Yaskawa INFORM job: ramp_standing_planes_program.JBI

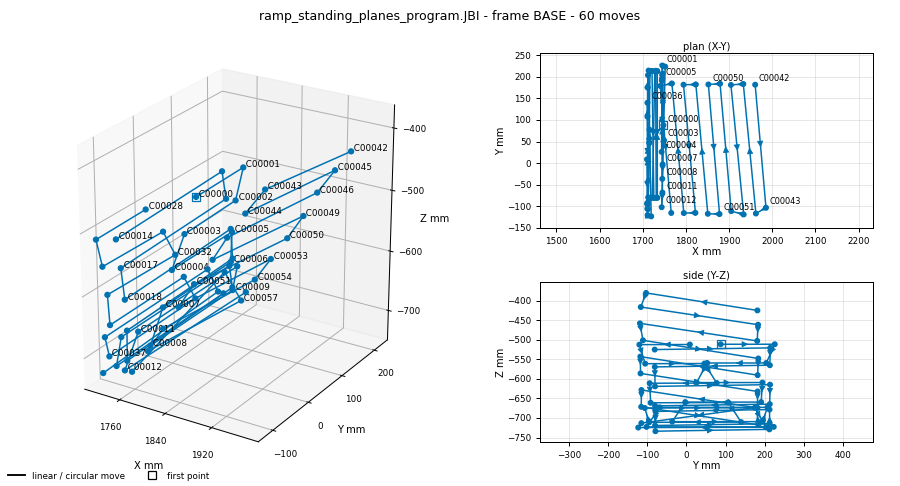
[picture p0: tool path of ramp_standing_planes_program.JBI in frame BASE, 60 of 65 moves have a stored position in this frame; points joined in program order, loops and branches not executed]
/JOB
//NAME ramp_standing_planes_program
//POS
///NPOS 60,0,60,0,0,0
///TOOL 0
///POSTYPE BASE
///RECTAN
///RCONF 0,0,0,0,0,0,0,0,0,0,0,0,0,0,0,0,0,0,0,0,0,0,0,0
C00000=1747.833676,87.707513,-511.371116,5.000000,-89.957822,175.000000
C00001=1745.440097,225.996535,-511.342791,5.000000,-89.957822,175.000000
C00002=1744.923440,204.207688,-559.299641,5.000000,-89.957822,175.000000
C00003=1749.154270,53.149469,-559.329393,5.000000,-89.957822,175.000000
C00004=1743.721814,26.039255,-609.339304,5.000000,-89.957822,175.000000
C00005=1744.348289,194.565765,-609.302177,5.000000,-89.957822,175.000000
C00006=1744.187925,191.095267,-659.303065,5.000000,-89.957822,175.000000
C00007=1746.082813,-2.901127,-659.343877,5.000000,-89.957822,175.000000
C00008=1745.263776,-36.374100,-709.351778,5.000000,-89.957822,175.000000
C00009=1745.079107,194.848338,-709.301607,5.000000,-89.957822,175.000000
C00010=1746.036638,207.361004,-672.695654,180.000000,-60.000000,0.000000
C00011=1745.574257,-68.103268,-672.755927,180.000000,-60.000000,0.000000
C00012=1743.877002,-102.062921,-722.764579,180.000000,-60.000000,0.000000
C00013=1752.018887,223.400139,-722.687777,180.000000,-60.000000,0.000000
C00014=1718.533268,-81.118931,-524.973339,5.000000,-87.037114,175.000000
C00015=1713.684878,214.380906,-520.671837,5.000000,-87.037114,175.000000
C00016=1721.540048,213.468866,-565.028354,5.000000,-87.037114,175.000000
C00017=1725.758225,-80.815821,-569.343755,5.000000,-87.037114,175.000000
C00018=1731.242809,-80.197878,-619.123216,5.000000,-87.037114,175.000000
C00019=1729.852338,213.811139,-614.665704,5.000000,-87.037114,175.000000
C00020=1733.681143,213.171353,-664.550241,5.000000,-87.037114,175.000000
C00021=1733.797506,-80.066986,-669.061826,5.000000,-87.037114,175.000000
C00022=1733.019581,-80.164547,-719.176447,5.000000,-87.037114,175.000000
C00023=1733.370862,212.848816,-714.644124,5.000000,-87.037114,175.000000
C00024=1727.945778,212.635262,-678.398521,180.000000,-60.000000,0.000000
C00025=1722.359725,-78.980421,-683.180255,180.000000,-60.000000,0.000000
C00026=1712.658875,-79.296819,-733.760083,180.000000,-60.000000,0.000000
C00027=1716.885173,212.264276,-729.049569,180.000000,-60.000000,0.000000
C00028=1709.955725,8.794869,-512.045023,5.000000,-89.491817,175.000000
C00029=1711.306908,-120.321693,-512.369923,5.000000,-89.491817,175.000000
C00030=1710.700045,-105.520124,-561.084797,5.000000,-89.491817,175.000000
C00031=1715.144631,46.230498,-560.649434,5.000000,-89.491817,175.000000
C00032=1715.725129,77.457805,-610.564946,5.000000,-89.491817,175.000000
C00033=1709.951896,-93.988220,-611.063481,5.000000,-89.491817,175.000000
C00034=1711.444659,-91.511088,-661.045915,5.000000,-89.491817,175.000000
C00035=1710.974292,107.455154,-660.530954,5.000000,-89.491817,175.000000
C00036=1710.807654,139.847878,-710.450052,5.000000,-89.491817,175.000000
C00037=1711.661647,-95.428769,-711.056349,5.000000,-89.491817,175.000000
C00038=1712.376345,-106.493392,-674.478476,180.000000,-60.000000,0.000000
C00039=1711.169902,174.896087,-673.754989,180.000000,-60.000000,0.000000
C00040=1712.211733,203.656058,-723.672846,180.000000,-60.000000,0.000000
C00041=1719.670531,-123.239544,-724.459608,180.000000,-60.000000,0.000000
C00042=1960.330006,181.614488,-424.835174,175.000000,-56.152488,-5.000000
C00043=1985.368889,-103.193855,-380.137392,175.000000,-56.152488,-5.000000
C00044=1962.016425,-116.674380,-416.148142,175.000000,-56.152488,-5.000000
C00045=1932.882821,183.234864,-461.360037,175.000000,-56.152488,-5.000000
C00046=1904.216477,181.050268,-502.826697,175.000000,-56.152488,-5.000000
C00047=1933.813388,-118.873277,-457.922429,175.000000,-56.152488,-5.000000
C00048=1904.866793,-111.166767,-501.336623,175.000000,-56.152488,-5.000000
C00049=1879.065944,183.890803,-547.736137,175.000000,-56.152488,-5.000000
C00050=1852.001340,182.186319,-590.380650,175.000000,-56.152488,-5.000000
C00051=1877.849575,-117.893555,-542.928603,175.000000,-56.152488,-5.000000
C00052=1850.711806,-117.345247,-586.010425,175.000000,-56.152488,-5.000000
C00053=1823.000964,182.124997,-632.081707,175.000000,-56.152488,-5.000000
C00054=1794.417051,181.587415,-673.959238,175.000000,-56.152488,-5.000000
C00055=1822.009926,-115.041980,-628.422180,175.000000,-56.152488,-5.000000
C00056=1795.135163,-115.591042,-671.443463,175.000000,-56.152488,-5.000000
C00057=1767.615554,184.356760,-717.746098,175.000000,-56.152488,-5.000000
C00058=1740.550659,178.708335,-672.936383,180.000000,-60.000000,0.000000
C00059=1766.041475,-115.340579,-713.149255,175.000000,-56.152488,-5.000000
///POSTYPE PULSE
///PULSE
EC00000=33792.0
EC00001=33792.0
EC00002=33792.0
EC00003=33792.0
EC00004=33792.0
EC00005=33792.0
EC00006=33792.0
EC00007=33792.0
EC00008=33792.0
EC00009=33792.0
EC00010=33792.0
EC00011=33792.0
EC00012=33792.0
EC00013=33792.0
EC00014=125952.0
EC00015=125952.0
EC00016=125952.0
EC00017=125952.0
EC00018=125952.0
EC00019=125952.0
EC00020=125952.0
EC00021=125952.0
EC00022=125952.0
EC00023=125952.0
EC00024=125952.0
EC00025=125952.0
EC00026=125952.0
EC00027=125952.0
EC00028=218112.0
EC00029=218112.0
EC00030=218112.0
EC00031=218112.0
EC00032=218112.0
EC00033=218112.0
EC00034=218112.0
EC00035=218112.0
EC00036=218112.0
EC00037=218112.0
EC00038=218112.0
EC00039=218112.0
EC00040=218112.0
EC00041=218112.0
EC00042=310272.0
EC00043=310272.0
EC00044=310272.0
EC00045=310272.0
EC00046=310272.0
EC00047=310272.0
EC00048=310272.0
EC00049=310272.0
EC00050=310272.0
EC00051=310272.0
EC00052=310272.0
EC00053=310272.0
EC00054=310272.0
EC00055=310272.0
EC00056=310272.0
EC00057=310272.0
EC00058=310272.0
EC00059=310272.0
//INST
///DATE 2023/08/13 13:32
///ATTR SC,RW,RJ
////FRAME BASE
///GROUP1 RB1,ST1
NOP
MOVJ P009 EX000 VJ=15.00
MOVJ C00000 EC00000 VJ=15.0
CALL JOB:SPYON
MOVL C00001 EC00001 V=150.0
MOVL C00002 EC00002 V=150.0
MOVL C00003 EC00003 V=150.0
MOVL C00004 EC00004 V=150.0
MOVL C00005 EC00005 V=150.0
MOVL C00006 EC00006 V=150.0
MOVL C00007 EC00007 V=150.0
MOVL C00008 EC00008 V=150.0
MOVL C00009 EC00009 V=150.0
MOVL C00010 EC00010 V=150.0
MOVL C00011 EC00011 V=150.0
MOVL C00012 EC00012 V=150.0
MOVL C00013 EC00013 V=150.0
CALL JOB:SPYOF
MOVJ P009 VJ=15.00
MOVJ C00014 EC00014 VJ=15.0
CALL JOB:SPYON
MOVL C00015 EC00015 V=150.0
MOVL C00016 EC00016 V=150.0
MOVL C00017 EC00017 V=150.0
MOVL C00018 EC00018 V=150.0
MOVL C00019 EC00019 V=150.0
MOVL C00020 EC00020 V=150.0
MOVL C00021 EC00021 V=150.0
MOVL C00022 EC00022 V=150.0
MOVL C00023 EC00023 V=150.0
MOVL C00024 EC00024 V=150.0
MOVL C00025 EC00025 V=150.0
MOVL C00026 EC00026 V=150.0
MOVL C00027 EC00027 V=150.0
CALL JOB:SPYOF
MOVJ P009 VJ=15.00
MOVJ C00028 EC00028 VJ=15.0
CALL JOB:SPYON
MOVL C00029 EC00029 V=150.0
MOVL C00030 EC00030 V=150.0
MOVL C00031 EC00031 V=150.0
MOVL C00032 EC00032 V=150.0
MOVL C00033 EC00033 V=150.0
MOVL C00034 EC00034 V=150.0
MOVL C00035 EC00035 V=150.0
MOVL C00036 EC00036 V=150.0
MOVL C00037 EC00037 V=150.0
MOVL C00038 EC00038 V=150.0
MOVL C00039 EC00039 V=150.0
MOVL C00040 EC00040 V=150.0
MOVL C00041 EC00041 V=150.0
CALL JOB:SPYOF
MOVJ P009 VJ=15.00
MOVJ C00042 EC00042 VJ=15.0
CALL JOB:SPYON
MOVL C00043 EC00043 V=150.0
MOVL C00044 EC00044 V=150.0
MOVL C00045 EC00045 V=150.0
MOVL C00046 EC00046 V=150.0
MOVL C00047 EC00047 V=150.0
MOVL C00048 EC00048 V=150.0
MOVL C00049 EC00049 V=150.0
MOVL C00050 EC00050 V=150.0
MOVL C00051 EC00051 V=150.0
MOVL C00052 EC00052 V=150.0
MOVL C00053 EC00053 V=150.0
MOVL C00054 EC00054 V=150.0
MOVL C00055 EC00055 V=150.0
MOVL C00056 EC00056 V=150.0
MOVL C00057 EC00057 V=150.0
MOVL C00058 EC00058 V=150.0
MOVL C00059 EC00059 V=150.0
CALL JOB:SPYOF
MOVJ P009 VJ=15.00
END
